FUNCTION TryConvert_UINT_TO_DT : BOOL
VAR_INPUT
	in : UINT;
	out : REFERENCE TO DT;
END_VAR

out := UINT_TO_DT(in);
TryConvert_UINT_TO_DT := TRUE;

END_FUNCTION

(* stored: Version 1.1.0.1, ProductVersion 3.1.4024.12
   POU TryConvert_UINT_TO_DT: Id {19864222-5f43-499f-bce0-2b7381fe660a}, SpecialFunc None *)
